FUNCTION_BLOCK T_InitModeManagerWithState EXTENDS T_UnitTestBase
VAR
  stateModule : T_MockStateModule;
  modeManager : T_ModeManager(stateModule);
  
  actual, expected : UINT;
END_VAR

//arrange
stateModule._currentState := 5;

//act

actual := TO_UINT(modeManager._state.CurrentState);
expected := 5;
//assert
assertion.AssertEquals_UDINT(actual, expected , 'actual := modeManager._state');
TestFinished();

END_FUNCTION_BLOCK

(* stored: Version 1.1.0.1, ProductVersion 3.1.4024.12
   POU T_InitModeManagerWithState: Id {2953af92-bc5e-426d-b2e3-d4ccc528258d}, SpecialFunc None *)
